// TIA Portal V20 export
VAR_GLOBAL   // PLC tag table "CITI"
END_VAR
